INTERFACE ISafetyComponent EXTENDS ITcoComponent

METHOD Resume
VAR_INPUT
END_VAR
END_METHOD

METHOD ServiceRequest
VAR_INPUT
END_VAR
END_METHOD

END_INTERFACE

(* stored: Version 1.1.0.1
   Itf ISafetyComponent: Id {fecdc336-73fb-440a-8842-f0e77c2c38d3}
   Method Resume: Id {feac7e84-aeef-4ec9-84fb-5503ef8ecb64}
   Method ServiceRequest: Id {bf695cdc-78a4-4e4b-948e-770786cec75d} *)
